INTERFACE ITF_BaseExecutiveElement_HMI_Connector EXTENDS ITF_BaseComplexElement_HMI_Connector

END_INTERFACE

(* stored: Version 1.1.0.1
   Itf ITF_BaseExecutiveElement_HMI_Connector: Id {68ea5254-c6f9-0b12-28dd-4a241e11bb89} *)
